// TIA Portal V17 export
// export: Created 2023-02-26T22:59:52.4093192Z, ExportSetting WithDefaults, DisplayName Totally Integrated Automation Portal, DisplayVersion V17, DisplayName TIA Portal Openness, DisplayVersion V17, DisplayName TIA Portal Version Control Interface, DisplayVersion V17, DisplayName TIA Portal Test Suite Advanced, DisplayVersion V17, DisplayName STEP 7 Professional, DisplayVersion V17, DisplayName SIMATIC Energy Suite, DisplayVersion V17, DisplayName STEP 7 Safety, DisplayVersion V17, DisplayName WinCC Professional, DisplayVersion V17
DATA_BLOCK "LOG_CountMode_DB_2"   // DB33
VERSION : 0.1
// stored: AutoNumber true, InstanceOfName LOG_CountMode, InstanceOfType FB
"LOG_CountMode"
   // VAR_INPUT
   //    "StartLine/StopLine" : Bool;
   //    Mode : Bool;
   // END_VAR
   // VAR_IN_OUT
   //    QMode : UDInt;
   // END_VAR
   // VAR
   //    P_Mode : Bool;
   // END_VAR
BEGIN
END_DATA_BLOCK
